(*
Nazwa:			P11_RollerScrewer
Opis:			Stacja zakręcarki rolkowej
Wersja:			v0.1
Data:			2018-10-10
Autor:			DP
Urzadzenia:		
Konfiguracja:	
Info:

*)
PROGRAM P11_RollerScrewer
VAR_INPUT

END_VAR
VAR
	(*********Zakręcarka rolkowa******)
	fbRollerScrewer: FB_RollerScrewer;		// Blok sterowania zakręcarką rolkową
	eRollerScrewerState: 			E_Station;						// Stan zakręcarki
	eRollerScrewerRunningState: 	E_RollerScrewer;				// Stan zakręcarki
	fbRollerScrewerState: 			FB_State;
	
	(************Chwytak*************)	
	fbRollerScrewerCatchStation						: FB_CatchStation;		
	eRollerScrewerCatchState						: E_Station;            
	eRollerScrewerCatchRunningState					: E_CatchStationState;  
	fbRollerScrewerCatchState						: FB_State;
	
	(************Szlaban*************)		
	fbRollerScrewerGate								: FB_SpringGateV2;

	
	// WEJŚĆIA I WYJŚCIA SPRZĘTOWE
	IbRollerScrewerHeightEncoderSetCDone			AT %I*: BOOL;
	IudiRollerScrewerHeightEncoderCV          		AT %I*: UDINT;
	QbRollerScrewerHeightEncoderSetC 				AT %Q*: BOOL;
	QudiRollerScrewerHeightEncoderSetCV       		AT %Q*: UDINT;

	QbRollerScrewerCatchHeightUpCmd 				AT %Q*: BOOL; 		
	QbRollerScrewerCatchHeightDownCmd 				AT %Q*: BOOL; 		
	IbRollerScrewerCatchHeightEncoderSetCDone		AT %I*: BOOL;
	IudiRollerScrewerCatchHeightEncoderCV          	AT %I*: UDINT;
	QbRollerScrewerCatchHeightEncoderSetC 			AT %Q*: BOOL;
	QudiRollerScrewerCatchHeightEncoderSetCV       	AT %Q*: UDINT;

	QABPneumaticRollerScrewerValveCoils 			AT %Q* 	: ARRAY[1..5] OF BYTE;	
	IuiPneumaticRollerScrewerState					AT %I* 	: UINT;	


	IbRollerScrewerFuseFB1OK						AT %I*	:BOOL;		
	IbRollerScrewerFuseRollerScrewerOK				AT %I*	:BOOL;		
	IbRollerScrewerFuseRollerScrewerCatchOK			AT %I*	:BOOL;		
	IbRollerScrewerPowerSupplyOK					AT %I*	:BOOL;
	//GVL_IO_SAFETY.IbSafetyRelayRC40	 			AT %I*  :BOOL;	
	IbRollerScrewerDoors1Open 						AT %I*	:BOOL;		
	IbRollerScrewerCycleStartStopButton				AT %I*	:BOOL;	
	IbRollerScrewerCompressedAirOK 					AT %I*	:BOOL;		
	IbRollerScrewerUnPressedTopSensor 				AT %I*	:BOOL;	
	IbRollerScrewerRollsUnPressedSensor 			AT %I*	:BOOL; 

	IbRollerScrewerCatchSensorOpened				AT %I*	:BOOL; 
	IbRollerScrewerDoors2Open 						AT %I*	:BOOL;			
	IbRollerScrewerCapPuttedSensor 					AT %I*	:BOOL;	
	QbRollerScrewerGreenSignalizationLamp 			AT %Q* : BOOL;			
	QbRollerScrewerRedSignalizationLamp 			AT %Q* : BOOL;				
	QbRollerScrewerWhiteSignalizationLamp 			AT %Q* : BOOL;						
	QbRollerScrewerYellowSignalizationLamp 			AT %Q* : BOOL;							
	QbRollerScrewerHeightMotorUp 					AT %Q*: BOOL;		
	QbRollerScrewerHeightMotorDown 					AT %Q*: BOOL;			
	
	QbRollerScrewerGate								: BOOL; 	
	QbRollerScrewerPressingTopActuator				: BOOL; 	
	QbRollerScrewerPressingRollsActuator			: BOOL; 	
	QbRollerScrewerCatchActuator					: BOOL; 

	QnRollerScrewerFrontTorqueLimit 				AT %Q*: UINT; 
	QnRollerScrewerRearTorqueLimit 					AT %Q*: UINT; 
	IrRollerScrewerRearActualMotorTemperature 		AT %I*: REAL; 
	IrRollerScrewerFrontActualMotorTemperature 		AT %I*: REAL; 

	(*RFID*)
	//Przed
	bReadedCard 										: BOOL;				
	nReadedCard											: ULINT;	
	fbReader   											: FB_IfmIoLinkRfid;
	AusiReaderInputData  								AT %I* : ARRAY[0..27] OF USINT;
	IbReaderTagPresent									AT %I* : BOOL;
	IBReaderErrorValue									AT %I* : BYTE;
	IbReaderCmdEnd										AT %I* : BOOL;
	IBReaderDataCounterIn								AT %I* : BYTE;
	IbReaderCmdStartAck									AT %I* : BOOL;
	IbReaderCmdStart									AT %Q* : BOOL;
	IBReaderCmmandValue									AT %Q* : BYTE;
	IBReaderDataCounterOut								AT %Q* : BYTE;
	AusiReaderOutputData  								AT %Q* : ARRAY[0..27] OF USINT;	


	TimerRollerScrewerEnable: TOF;
	TimerRollerScrewerCatchEnable: TOF;
	tonLidPuttedCheckEnable: TON;	
	rtEnable: R_TRIG;	
	
	(*Wykres dozowania*)
	fbRollerScrewingChart: FB_WriteDataToArrayString;

	rtStartRollerScrewing: R_TRIG;
	lrRollerScrewerAxisStartPosition: LREAL;

	tonRollerScrewerCatchSensorOpened: TON;
	


END_VAR

aPowerSupply();
aButtons();
aPneumatics();
aRFID();
aRFID_FB();
aSafety();
aSignalization();
aLimits();
a1_Gate();
a1_GateTime();
a2_RollerScrewer();
aWarnings();

(*** SKALOWANIE WARTOŚCI ZAKRĘCANIA Z Nm na % ***)
(* Wersja w Nm fbRollerScrewer.iScrewerSetTorque 
:=LREAL_TO_INT( 
													(lrRollerScrewingTightTorque/(INT_TO_LREAL(iPackageCapDiameter)*0.0633))*100
												 );*)
												 
fbRollerScrewer.iScrewerSetTorque :=LREAL_TO_INT(lrRollerScrewingTightTorque);												 
(*** KONIEC SKALOWANIE WARTOŚCI ZAKRĘCANIA Z Nm na % ***)

(*SYMULACJA CZUJNIKÓW*)
tonRollerScrewerCatchSensorOpened(IN:=NOT QbRollerScrewerCatchActuator, PT:=T#10MS);//bylo 300


(* BAZOWANIE - ZMIAN*)
tonLidPuttedCheckEnable(IN:=fbRollerScrewer.bEnable,PT:=T#5S); (*Dodany ton bo Wizka zjebnie wgrywa zmienne, najpierw włacza Enabla a potem dopiero wybiera recepture*)
//rtEnable(CLK:=fbRollerScrewer.bEnable,Q=>);
rtEnable(CLK:=tonLidPuttedCheckEnable.Q,Q=>);
// IF rtEnable.Q AND eMachineState>=E_MachineState.eReady AND eMachineState<>E_MachineState.eHardError  THEN
// 	VIS.bRollerScrewerCatchHeightSet:=TRUE;
// 	//VIS.bRollerScrewerHeightSet:=TRUE;
// ELSIF fbRollerScrewer.eState=E_Station.eHomingDone OR eMachineState=E_MachineState.eHardError THEN
//  	VIS.bRollerScrewerHeightSet:=FALSE;
// ELSIF  fbRollerScrewerCatchStation.eState=E_Station.eHomingDone OR eMachineState=E_MachineState.eHardError THEN
// 	VIS.bRollerScrewerHeightSet:=TRUE; //Zmiana LU208
// 	VIS.bRollerScrewerCatchHeightSet:=FALSE;
// END_IF
(*KONIEC BAZOWANIE - ZMIANA*)


(********* GENEROWANIE STANU STACJI DO WIZKI**********)
// fbRollerScrewerState(
// 	eState:=eRollerScrewerState , 
// 	bRun:=bStartRollerScrewing OR VIS.bManualStartRollerScrew,	
// 	eRollerScrewerRunningState:=eRollerScrewerRunningState , 
// 	sStateDesc=> VIS.sRollerScrewerState,
// 	iState=>VIS.iRollerScrewerState);
//fbRollerScrewerCatchState(
//	eState:=eRollerScrewerCatchState , 
//	bRun:=bRollerScrewerCatch,	
//	eCatchRunningState:=eRollerScrewerCatchRunningState , 
//	sStateDesc=> VIS.sRollerScrewerCatchState,
//	iState=>VIS.iRollerScrewerCatchState);	
(***** KONIEC GENEROWANIE STANU STACJI DO WIZKI*******)

(*Opoznienie wyłączanie enabla*)
TimerRollerScrewerEnable 		(IN:=bRollerScrewerEnable  AND NOT bChangeover , PT:=T#2S);
TimerRollerScrewerCatchEnable 	(IN:=bRollerScrewerEnable  AND NOT bChangeover , PT:=T#4S);
{warning 'Zmienione włączenie/wyłączanie rolkowej do testów'}

(*Przypisywanie wartości*)
IF fbRollerScrewerCatchStation.lrHeightMotorCV+24 <= 65 THEN //Warrtość minimalna stacji zakrecarki rolkowej
	fbRollerScrewer.lrMinHeight := 60; //Warrtość minimalna stacji zakrecarki rolkowej
ELSE	//Jezeli ponad minimalną to minimalna jest wartościa chwytaka
	fbRollerScrewer.lrMinHeight:=fbRollerScrewerCatchStation.lrHeightMotorCV+10; 
END_IF

(********KASOWANIE ROZKAZÓW CYKLI*********)
IF fbRollerScrewer.bCycleDone AND bManualMode THEN
	VIS_RS.bRollerScrewerRun := FALSE;
END_IF
(*****KONIEC KASOWANIA ROZKAZÓW CYKLI*****)

ACTION a1_Gate:
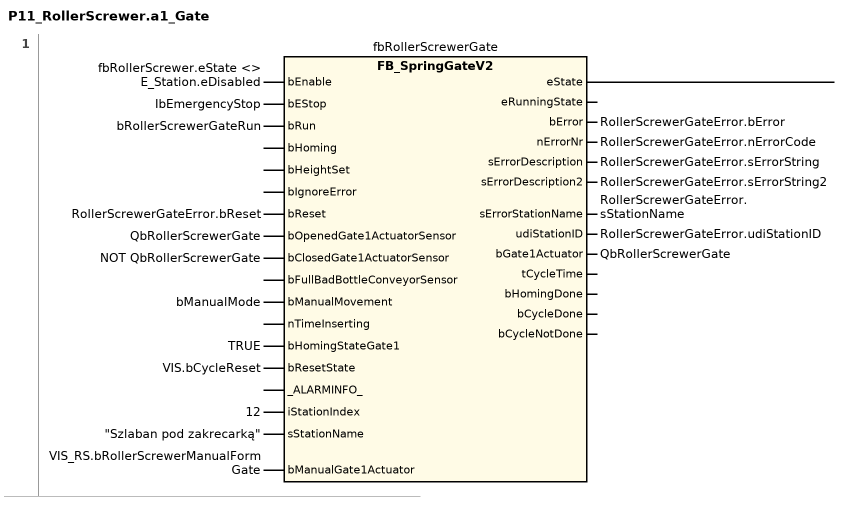
// NETWORK 1
fbRollerScrewerGate(
    bEnable := fbRollerScrewer.eState <> E_Station.eDisabled,
    bEStop := IbEmergencyStop,
    bRun := bRollerScrewerGateRun,
    bReset := RollerScrewerGateError.bReset,
    bOpenedGate1ActuatorSensor := QbRollerScrewerGate,
    bClosedGate1ActuatorSensor := NOT QbRollerScrewerGate,
    bManualMovement := bManualMode,
    bHomingStateGate1 := TRUE,
    bResetState := VIS.bCycleReset,
    iStationIndex := 12,
    sStationName := "Szlaban pod zakrecarką",
    bManualGate1Actuator := VIS_RS.bRollerScrewerManualFormGate,
    bError => RollerScrewerGateError.bError,
    nErrorNr => RollerScrewerGateError.nErrorCode,
    sErrorDescription => RollerScrewerGateError.sErrorString,
    sErrorDescription2 => RollerScrewerGateError.sErrorString2,
    sErrorStationName => RollerScrewerGateError.sStationName,
    udiStationID => RollerScrewerGateError.udiStationID,
    bGate1Actuator => QbRollerScrewerGate); // FB_SpringGateV2
END_ACTION

ACTION a1_GateTime:

fbRollerScrewerGate.nTimeInserting	:=	300;
END_ACTION

ACTION a2_RollerScrewer:
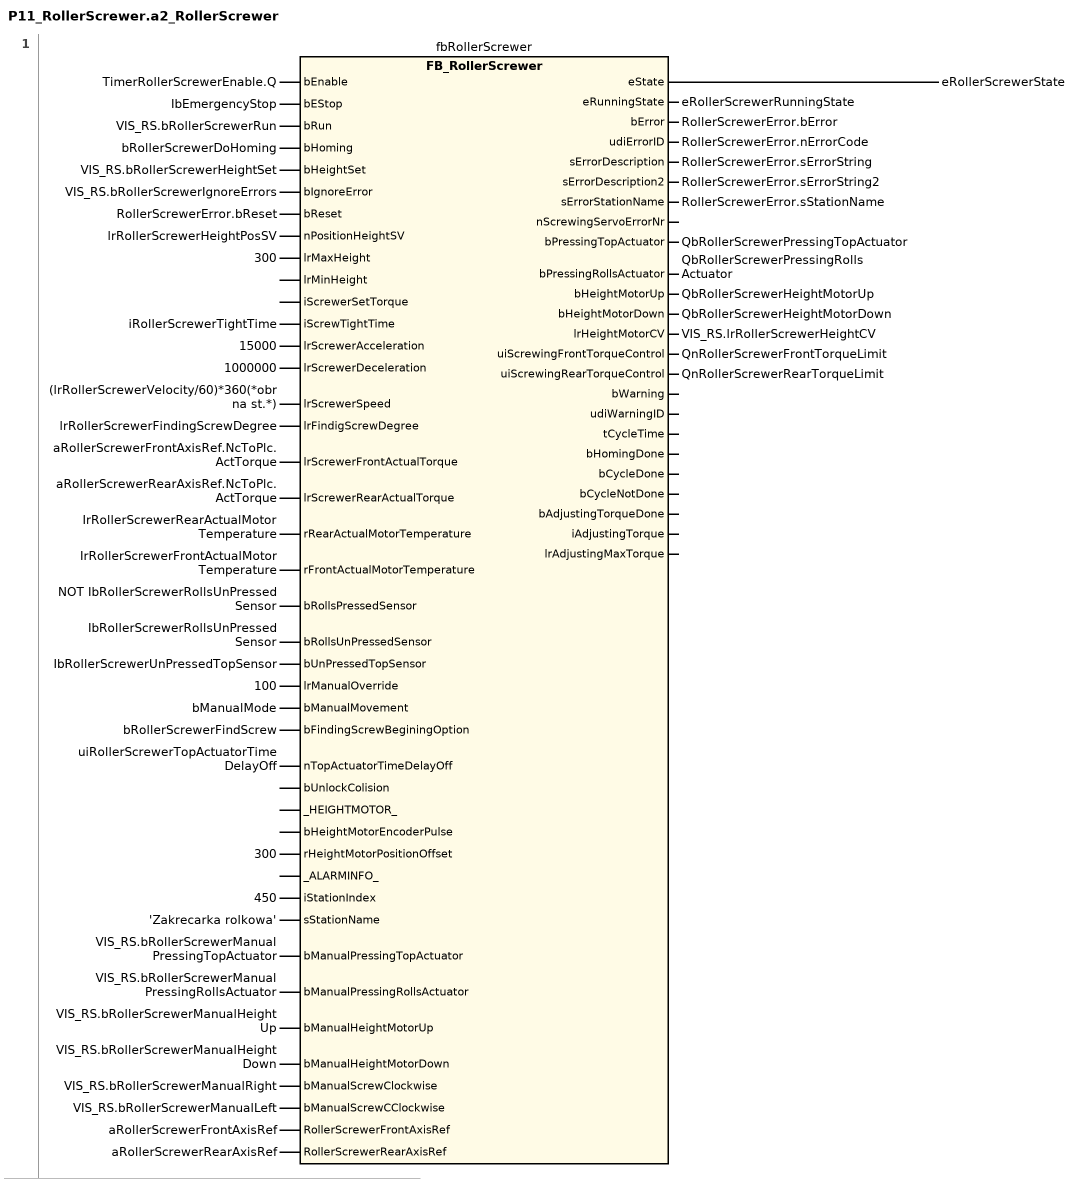
// NETWORK 1
fbRollerScrewer(
    bEnable := TimerRollerScrewerEnable.Q,
    bEStop := IbEmergencyStop,
    bRun := VIS_RS.bRollerScrewerRun,
    bHoming := bRollerScrewerDoHoming,
    bHeightSet := VIS_RS.bRollerScrewerHeightSet,
    bIgnoreError := VIS_RS.bRollerScrewerIgnoreErrors,
    bReset := RollerScrewerError.bReset,
    nPositionHeightSV := lrRollerScrewerHeightPosSV,
    lrMaxHeight := 300,
    iScrewTightTime := iRollerScrewerTightTime,
    lrScrewerAcceleration := 15000,
    lrScrewerDeceleration := 1000000,
    lrScrewerSpeed := (lrRollerScrewerVelocity/60)*360(*obr na st.*),
    lrFindigScrewDegree := lrRollerScrewerFindingScrewDegree,
    lrScrewerFrontActualTorque := aRollerScrewerFrontAxisRef.NcToPlc.ActTorque,
    lrScrewerRearActualTorque := aRollerScrewerRearAxisRef.NcToPlc.ActTorque,
    rRearActualMotorTemperature := IrRollerScrewerRearActualMotorTemperature,
    rFrontActualMotorTemperature := IrRollerScrewerFrontActualMotorTemperature,
    bRollsPressedSensor := NOT IbRollerScrewerRollsUnPressedSensor,
    bRollsUnPressedSensor := IbRollerScrewerRollsUnPressedSensor,
    bUnPressedTopSensor := IbRollerScrewerUnPressedTopSensor,
    lrManualOverride := 100,
    bManualMovement := bManualMode,
    bFindingScrewBeginingOption := bRollerScrewerFindScrew,
    nTopActuatorTimeDelayOff := uiRollerScrewerTopActuatorTimeDelayOff,
    rHeightMotorPositionOffset := 300,
    iStationIndex := 450,
    sStationName := 'Zakrecarka rolkowa',
    bManualPressingTopActuator := VIS_RS.bRollerScrewerManualPressingTopActuator,
    bManualPressingRollsActuator := VIS_RS.bRollerScrewerManualPressingRollsActuator,
    bManualHeightMotorUp := VIS_RS.bRollerScrewerManualHeightUp,
    bManualHeightMotorDown := VIS_RS.bRollerScrewerManualHeightDown,
    bManualScrewClockwise := VIS_RS.bRollerScrewerManualRight,
    bManualScrewCClockwise := VIS_RS.bRollerScrewerManualLeft,
    RollerScrewerFrontAxisRef := aRollerScrewerFrontAxisRef,
    RollerScrewerRearAxisRef := aRollerScrewerRearAxisRef,
    eRunningState => eRollerScrewerRunningState,
    bError => RollerScrewerError.bError,
    udiErrorID => RollerScrewerError.nErrorCode,
    sErrorDescription => RollerScrewerError.sErrorString,
    sErrorDescription2 => RollerScrewerError.sErrorString2,
    sErrorStationName => RollerScrewerError.sStationName,
    bPressingTopActuator => QbRollerScrewerPressingTopActuator,
    bPressingRollsActuator => QbRollerScrewerPressingRollsActuator,
    bHeightMotorUp => QbRollerScrewerHeightMotorUp,
    bHeightMotorDown => QbRollerScrewerHeightMotorDown,
    lrHeightMotorCV => VIS_RS.lrRollerScrewerHeightCV,
    uiScrewingFrontTorqueControl => QnRollerScrewerFrontTorqueLimit,
    uiScrewingRearTorqueControl => QnRollerScrewerRearTorqueLimit); // FB_RollerScrewer
eRollerScrewerState := fbRollerScrewer.eState;

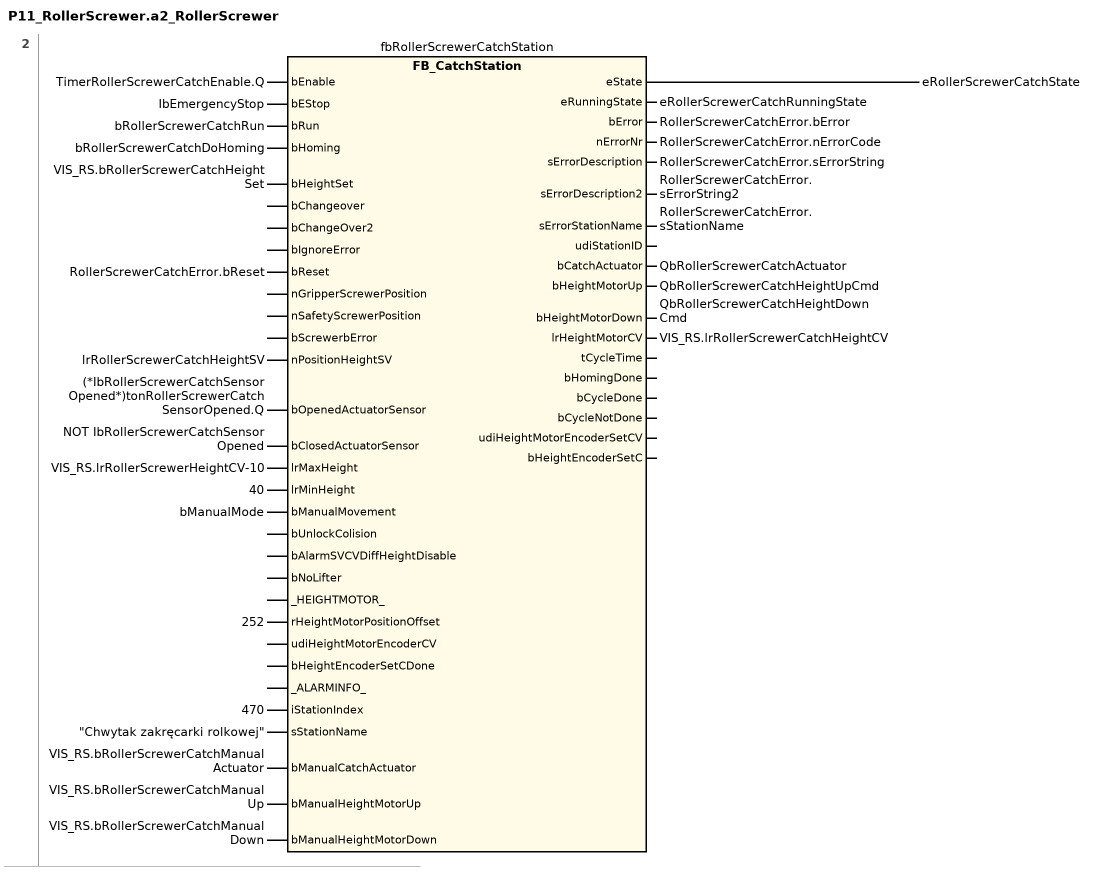
// NETWORK 2
fbRollerScrewerCatchStation(
    bEnable := TimerRollerScrewerCatchEnable.Q,
    bEStop := IbEmergencyStop,
    bRun := bRollerScrewerCatchRun,
    bHoming := bRollerScrewerCatchDoHoming,
    bHeightSet := VIS_RS.bRollerScrewerCatchHeightSet,
    bReset := RollerScrewerCatchError.bReset,
    nPositionHeightSV := lrRollerScrewerCatchHeightSV,
    bOpenedActuatorSensor := (*IbRollerScrewerCatchSensorOpened*)tonRollerScrewerCatchSensorOpened.Q,
    bClosedActuatorSensor := NOT IbRollerScrewerCatchSensorOpened,
    lrMaxHeight := VIS_RS.lrRollerScrewerHeightCV-10,
    lrMinHeight := 40,
    bManualMovement := bManualMode,
    rHeightMotorPositionOffset := 252,
    iStationIndex := 470,
    sStationName := "Chwytak zakręcarki rolkowej",
    bManualCatchActuator := VIS_RS.bRollerScrewerCatchManualActuator,
    bManualHeightMotorUp := VIS_RS.bRollerScrewerCatchManualUp,
    bManualHeightMotorDown := VIS_RS.bRollerScrewerCatchManualDown,
    eRunningState => eRollerScrewerCatchRunningState,
    bError => RollerScrewerCatchError.bError,
    nErrorNr => RollerScrewerCatchError.nErrorCode,
    sErrorDescription => RollerScrewerCatchError.sErrorString,
    sErrorDescription2 => RollerScrewerCatchError.sErrorString2,
    sErrorStationName => RollerScrewerCatchError.sStationName,
    bCatchActuator => QbRollerScrewerCatchActuator,
    bHeightMotorUp => QbRollerScrewerCatchHeightUpCmd,
    bHeightMotorDown => QbRollerScrewerCatchHeightDownCmd,
    lrHeightMotorCV => VIS_RS.lrRollerScrewerCatchHeightCV); // FB_CatchStation
eRollerScrewerCatchState := fbRollerScrewerCatchStation.eState;
END_ACTION

ACTION aButtons:

END_ACTION

ACTION aLimits:
(*
Nazwa:			aLimits
Opis:			Zabezpieczenia
Wersja:			v1.0
Data:			2023-11-24
Autor:			DP
Urzadzenia:		
Zmiany:	

Info:
*)

(**** Limity i zabezpieczenia***)
END_ACTION

ACTION aPneumatics:
// Do podpięcia według kolejności
QbRollerScrewerGate						;	
QbRollerScrewerPressingTopActuator		;
QbRollerScrewerPressingRollsActuator	;
QbRollerScrewerCatchActuator			;
;


(*************************** CapPusher EB1 **************************************)
// Wyspa 1 - dozowanie
IuiPneumaticRollerScrewerState;
QABPneumaticRollerScrewerValveCoils[1].0 := NOT QbRollerScrewerGate;
QABPneumaticRollerScrewerValveCoils[1].1 := QbRollerScrewerGate;
QABPneumaticRollerScrewerValveCoils[1].2 ;//
QABPneumaticRollerScrewerValveCoils[1].3 ;//
QABPneumaticRollerScrewerValveCoils[1].4 ;//
QABPneumaticRollerScrewerValveCoils[1].5 ;//
QABPneumaticRollerScrewerValveCoils[1].6 ;//
QABPneumaticRollerScrewerValveCoils[1].7 ;//
QABPneumaticRollerScrewerValveCoils[2].0 := QbRollerScrewerPressingTopActuator;			
QABPneumaticRollerScrewerValveCoils[2].1 ;
QABPneumaticRollerScrewerValveCoils[2].2 ;
QABPneumaticRollerScrewerValveCoils[2].3 ;
QABPneumaticRollerScrewerValveCoils[2].4 := QbRollerScrewerPressingRollsActuator;
QABPneumaticRollerScrewerValveCoils[2].5 ;
QABPneumaticRollerScrewerValveCoils[2].6 := QbRollerScrewerCatchActuator;
QABPneumaticRollerScrewerValveCoils[2].7 ;										                                                        
(*********************Koniec CapPusher EB1 **************************************)
END_ACTION

ACTION aPowerSupply:


	//Dodane do głwnych
	IbRollerScrewerFuseFB1OK				;
	IbRollerScrewerFuseRollerScrewerOK		;
	IbRollerScrewerFuseRollerScrewerCatchOK	;
	IbRollerScrewerPowerSupplyOK			;
END_ACTION

ACTION aRFID:
(*Przepisanie bity wykrycia karty*)
bReadedCard 		:= IbReaderTagPresent AND fbReader.bCodeReaded;
nReadedCard 		:= DINT_TO_ULINT(fbReader.diReadedCode);
END_ACTION

ACTION aRFID_FB:
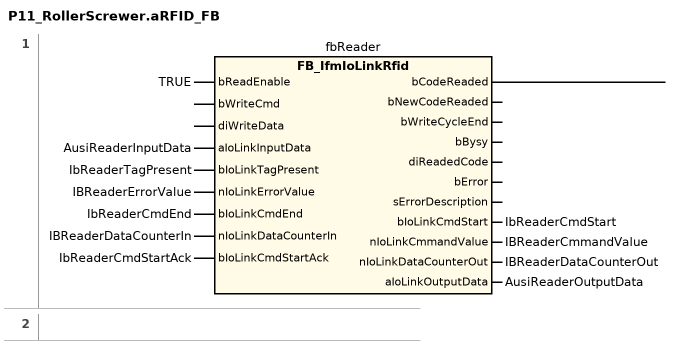
// NETWORK 1
fbReader(
    bReadEnable := TRUE,
    aIoLinkInputData := AusiReaderInputData,
    bIoLinkTagPresent := IbReaderTagPresent,
    nIoLinkErrorValue := IBReaderErrorValue,
    bIoLinkCmdEnd := IbReaderCmdEnd,
    nIoLinkDataCounterIn := IBReaderDataCounterIn,
    bIoLinkCmdStartAck := IbReaderCmdStartAck,
    bIoLinkCmdStart => IbReaderCmdStart,
    nIoLinkCmmandValue => IBReaderCmmandValue,
    nIoLinkDataCounterOut => IBReaderDataCounterOut,
    aIoLinkOutputData => AusiReaderOutputData); // FB_IfmIoLinkRfid

// NETWORK 2
END_ACTION

ACTION aRollerScrewerChartHMI:
(*Wykres zakręcarki rolkowej*)
rtStartRollerScrewing(CLK:=bStartRollerScrewing OR VIS.bManualStartRollerScrew, Q=>);
IF rtStartRollerScrewing.Q THEN (*Przy starcie zarkęcania, zapamiętywanie pozycji poczatkowej*)
	lrRollerScrewerAxisStartPosition := aRollerScrewerFrontAxisRef.NcToPlc.ActPos;
END_IF
 fbRollerScrewingChart(
	bWrite:= bStartRollerScrewing OR VIS.bManualStartRollerScrew, 
	nCycleTime:= 5, 
	lrData1:= aRollerScrewerFrontAxisRef.NcToPlc.ActPos - lrRollerScrewerAxisStartPosition, (*Zamiana st. na obr*)(*Odjęcie pozycji poczatkowej*) 
	lrData2:= aRollerScrewerFrontAxisRef.NcToPlc.ActTorque,// Wersja w Nm(aRollerScrewerFrontAxisRef.NcToPlc.ActTorque/100.0)*(INT_TO_LREAL(iPackageCapDiameter)*0.0633),  
	bData3:= QbRollerScrewerPressingRollsActuator, 
	bData4:= QbRollerScrewerPressingTopActuator,
	bData5:= FALSE,
	bData2B_ON:= FALSE,
	AsData=>VIS.AsChartRollerScrewing );
END_ACTION

ACTION aSafety:

// Dodać do P00_Alarms.aGeneralAlarms
	//IbCapPusherEmergencyStopButton0Pressed;
	//IbCapPusherEmergencyStopButton1Pressed;
	
(*
	IF IbCapPusherEmergencyStopButton0Pressed THEN
		GeneralAlarms.nErrorCode:=1;			
		GeneralAlarms.sErrorString:='Stop Awaryjny, sprawdź bezpieczeństwo, zresetuj przyciskiem na panelu | Naciśnięty przycisk awaryjny 1 na CapPusher';	
	ELSIF  IbCapPusherEmergencyStopButton1Pressed THEN
		GeneralAlarms.nErrorCode:=2;
		GeneralAlarms.sErrorString:='Stop Awaryjny, sprawdź bezpieczeństwo, zresetuj przyciskiem na panelu | Naciśnięty przycisk awaryjny 2 na CapPusher';	
*)	
	

// Dodać do miejsca gdzie są zamykane drzwi	
// lub zostawić tak jak jest
	IbRollerScrewerDoors1Open ;
	IbRollerScrewerDoors2Open ;
END_ACTION

ACTION aSignalization:
(*****Listwy LED*****)

QbRollerScrewerRedSignalizationLamp		:= INT_TO_BOOL(P00_Signalization.QiLineRedSignalizationLamp);
QbRollerScrewerGreenSignalizationLamp	:= INT_TO_BOOL(P00_Signalization.QiLineGreenSignalizationLamp);
QbRollerScrewerYellowSignalizationLamp	:= INT_TO_BOOL(P00_Signalization.QiLineBlueSignalizationLamp);
QbRollerScrewerWhiteSignalizationLamp ;

//QbCapPusherStartLamp	:= P00_Signalization.QbStartLamp;	   
//QbCapPusherResetLamp	:= P00_Signalization.QbResetLamp;
END_ACTION

ACTION aWarnings:
//Warning 0
//IF fbCapPusherFeeder.bWarning1 AND NOT CapSorterWarning[0].bWarning THEN
//	CapSorterWarning[0].bWarning										:=TRUE;
//	CapSorterWarning[0].udiWarningCode									:=41;
//	CapSorterWarning[0].sDescription									:='Sorter nasadek | Brak nasadek w zasobniku';
//ELSIF NOT fbCapPusherFeeder.bWarning1 THEN 
//	CapSorterWarning[0].bWarning										:=FALSE;
//	CapSorterWarning[0].bAcknowledge									:=FALSE;
//	VIS.uliWarningAcknowledge.27										:=FALSE;
//ELSIF CapSorterWarning[0].bAcknowledge THEN                               
//	CapSorterWarning[0].bAcknowledge									:=TRUE;
//END_IF
END_ACTION

END_PROGRAM

(* stored: Version 1.1.0.1, ProductVersion 3.1.4026.13
   POU P11_RollerScrewer: Id {0a92ffad-0950-45fd-9a25-21cfcd40ed2c}, SpecialFunc None
   Action a1_Gate: Id {8de00812-1921-4cbd-bec4-a77d50e869ee}
   Action a1_GateTime: Id {0edd0274-feee-440f-8449-761ca0bd0743}
   Action a2_RollerScrewer: Id {63df0243-f946-4e80-b65d-0dfa83801eb9}
   Action aButtons: Id {646b897d-8683-4954-81d8-7633bd59f9fd}
   Action aLimits: Id {c231477d-8758-49f4-9ebe-2ee0487d476f}
   Action aPneumatics: Id {4beaf567-0ee6-46d5-9bf4-05a4d71327cb}
   Action aPowerSupply: Id {0b0c340b-86d8-4b45-b394-d02193d75176}
   Action aRFID: Id {70eb136c-2a1f-431b-ae25-26552c9e0f85}
   Action aRFID_FB: Id {e0951058-ed40-4bd7-9c4d-fbdf13aae450}
   Action aRollerScrewerChartHMI: Id {46e933d6-3274-45f0-9ef7-ea3cc904cc75}
   Action aSafety: Id {4e2e1079-0ae8-4414-a7d5-052fc8c35171}
   Action aSignalization: Id {935f3be5-aaed-472a-9b02-86db9c7e28bb}
   Action aWarnings: Id {0e8fba99-20de-4977-85b5-96799a032f21} *)
